FUNCTION_BLOCK HandlingControl (* Basic FB with empty ECC *)
  (* Standard: 61499-2 *)
  (* Version 1.0, 2021-09-15, dorofeev *)
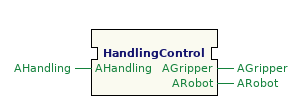
  SOCKETS
    AHandling : AHandling;
  END_SOCKETS
  PLUGS
    AGripper : AGripper;
    ARobot : ARobot;
  END_PLUGS
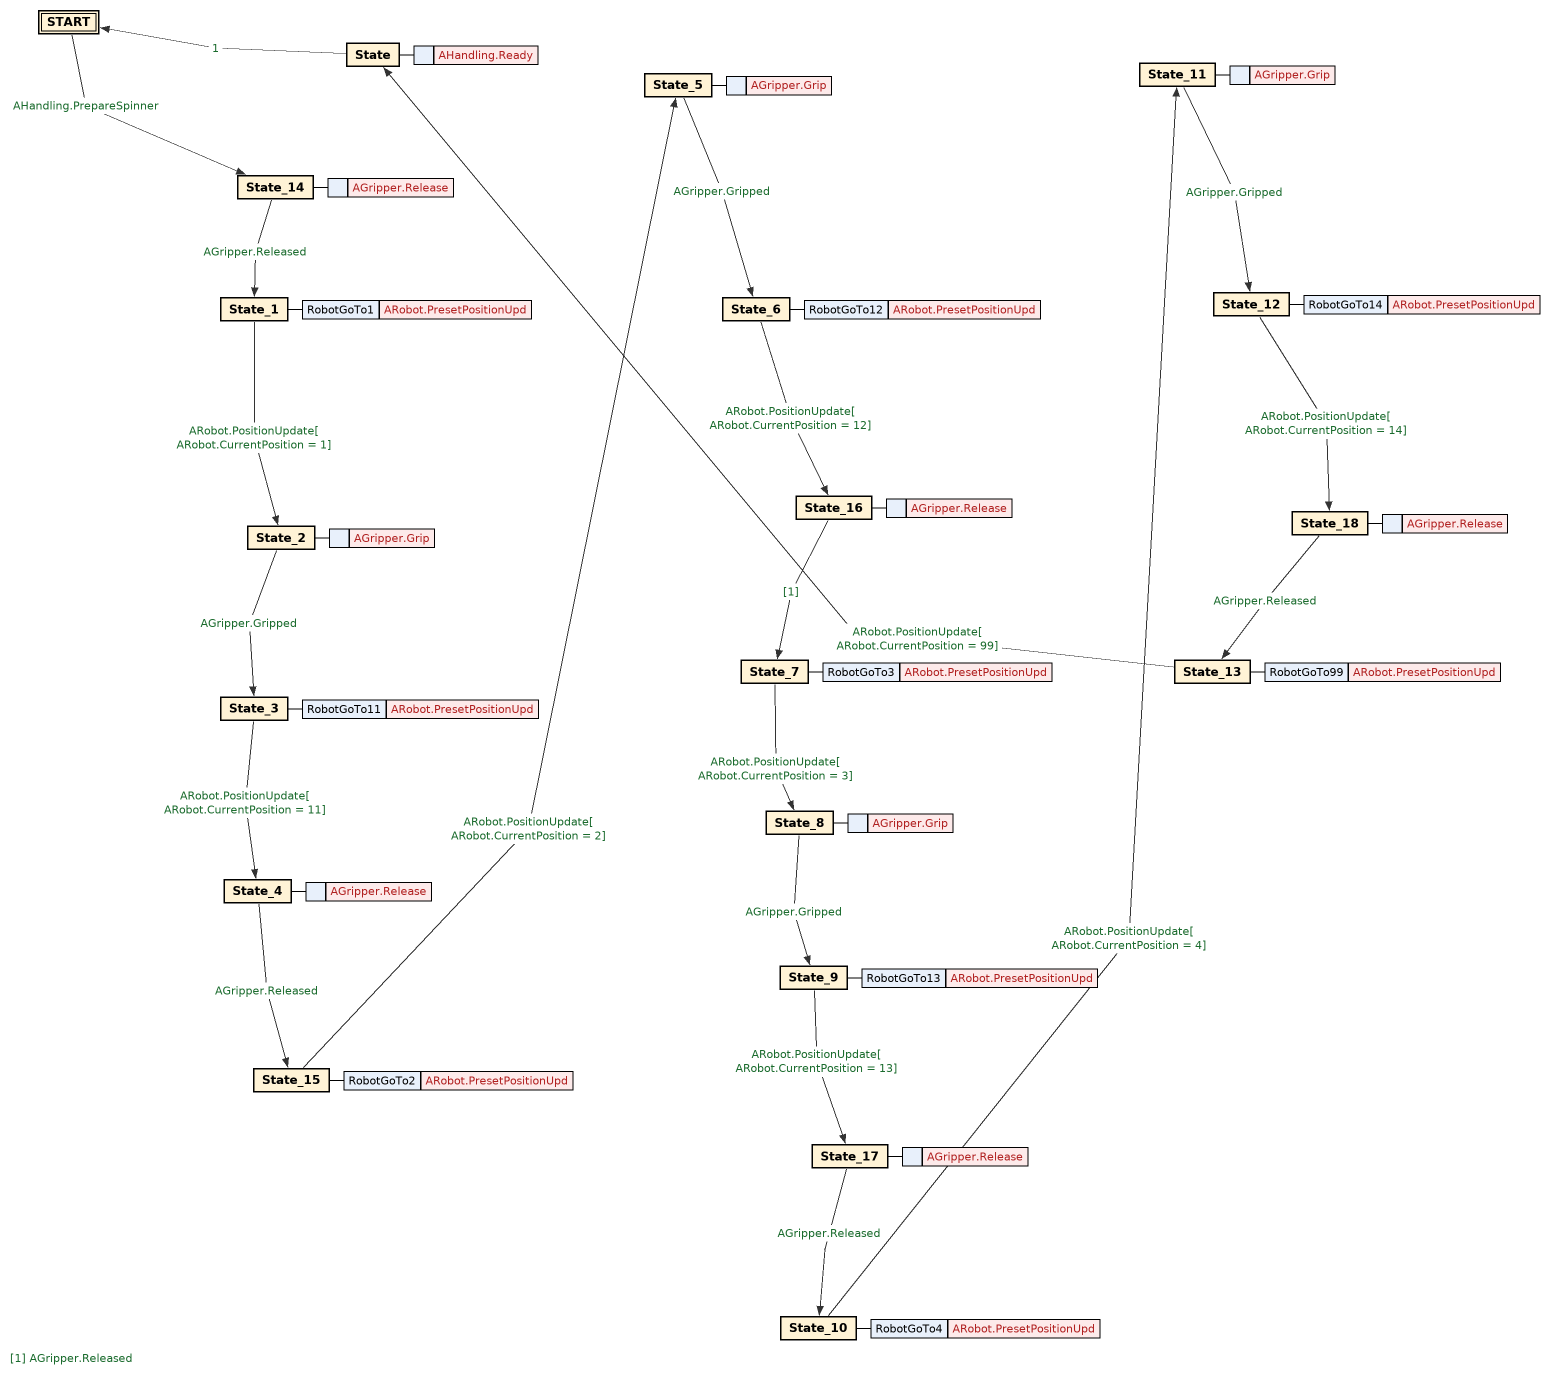
  EC_STATES
    START; (* Initial State *)
    State_1 : RobotGoTo1 -> ARobot.PresetPositionUpd;
    State_2 : -> AGripper.Grip;
    State_3 : RobotGoTo11 -> ARobot.PresetPositionUpd;
    State_4 : -> AGripper.Release;
    State_5 : -> AGripper.Grip;
    State_6 : RobotGoTo12 -> ARobot.PresetPositionUpd;
    State_7 : RobotGoTo3 -> ARobot.PresetPositionUpd;
    State_8 : -> AGripper.Grip;
    State_9 : RobotGoTo13 -> ARobot.PresetPositionUpd;
    State_10 : RobotGoTo4 -> ARobot.PresetPositionUpd;
    State_11 : -> AGripper.Grip;
    State_12 : RobotGoTo14 -> ARobot.PresetPositionUpd;
    State_13 : RobotGoTo99 -> ARobot.PresetPositionUpd;
    State : -> AHandling.Ready;
    State_14 : -> AGripper.Release;
    State_15 : RobotGoTo2 -> ARobot.PresetPositionUpd;
    State_16 : -> AGripper.Release;
    State_17 : -> AGripper.Release;
    State_18 : -> AGripper.Release;
  END_STATES
  EC_TRANSITIONS
    State_1 TO State_2 := ARobot.PositionUpdate[ARobot.CurrentPosition = 1];
    State_2 TO State_3 := AGripper.Gripped;
    State_3 TO State_4 := ARobot.PositionUpdate[ARobot.CurrentPosition = 11];
    State_5 TO State_6 := AGripper.Gripped;
    State_7 TO State_8 := ARobot.PositionUpdate[ARobot.CurrentPosition = 3];
    State_8 TO State_9 := AGripper.Gripped;
    State_10 TO State_11 := ARobot.PositionUpdate[ARobot.CurrentPosition = 4];
    State_11 TO State_12 := AGripper.Gripped;
    State_13 TO State := ARobot.PositionUpdate[ARobot.CurrentPosition = 99];
    State TO START := 1;
    START TO State_14 := AHandling.PrepareSpinner;
    State_14 TO State_1 := AGripper.Released;
    State_15 TO State_5 := ARobot.PositionUpdate[ARobot.CurrentPosition = 2];
    State_4 TO State_15 := AGripper.Released;
    State_6 TO State_16 := ARobot.PositionUpdate[ARobot.CurrentPosition = 12];
    State_16 TO State_7 := AGripper.Released;
    State_9 TO State_17 := ARobot.PositionUpdate[ARobot.CurrentPosition = 13];
    State_17 TO State_10 := AGripper.Released;
    State_12 TO State_18 := ARobot.PositionUpdate[ARobot.CurrentPosition = 14];
    State_18 TO State_13 := AGripper.Released;
  END_TRANSITIONS
  ALGORITHM RobotGoTo1 IN ST: (* New Algorithm *)
ARobot.PresetPosition := 1;
  END_ALGORITHM
  ALGORITHM RobotGoTo2 IN ST: (* New Algorithm *)
ARobot.PresetPosition := 2;
  END_ALGORITHM
  ALGORITHM RobotGoTo3 IN ST: (* New Algorithm *)
ARobot.PresetPosition := 3;
  END_ALGORITHM
  ALGORITHM RobotGoTo4 IN ST: (* New Algorithm *)
ARobot.PresetPosition := 4;
  END_ALGORITHM
  ALGORITHM RobotGoTo11 IN ST: (* New Algorithm *)
ARobot.PresetPosition := 11;
  END_ALGORITHM
  ALGORITHM RobotGoTo12 IN ST: (* New Algorithm *)
ARobot.PresetPosition := 12;
  END_ALGORITHM
  ALGORITHM RobotGoTo13 IN ST: (* New Algorithm *)
ARobot.PresetPosition := 13;
  END_ALGORITHM
  ALGORITHM RobotGoTo14 IN ST: (* New Algorithm *)
ARobot.PresetPosition := 14;
  END_ALGORITHM
  ALGORITHM RobotGoTo99 IN ST: (* New Algorithm *)
ARobot.PresetPosition := 99;
  END_ALGORITHM
END_FUNCTION_BLOCK
